# EPICS autosave request: xx_auto_userAve_settings.req
$(P)$(A).DESC
$(P)$(A).PREC
$(P)$(A).SCAN
$(P)$(A).INPB
$(P)$(A).A
